// TIA Portal V15.1 export
// export: Created 2024-05-17T05:38:34.4008009Z, ExportSetting WithDefaults, DisplayName Totally Integrated Automation Portal, DisplayVersion V15.1 Update 5, DisplayName TIA Portal Openness, DisplayVersion V15.1 Update 5, DisplayName SINAMICS Startdrive Advanced, DisplayVersion V15.1, DisplayName G130, G150, S120, S150, SINAMICS MV, S210, DisplayVersion V15.1, DisplayName G110M, G120, G120C, G120D, G120P, DisplayVersion V15.1, DisplayName STEP 7 Professional, DisplayVersion V15.1 Update 5, DisplayName STEP 7 Safety, DisplayVersion V15.1, DisplayName WinCC Professional, DisplayVersion V15.1 Update 5, DisplayName SIMATIC Visualization Architect, DisplayVersion V15.1
FUNCTION_BLOCK "LProcSel5SP"   // FB1712, FBD
TITLE = LProcSel5SP
{ S7_Optimized_Access := 'FALSE' }
AUTHOR : VCC
FAMILY : ProcEq
NAME : Sel5SP
VERSION : 0.1
// ================================================================================
// This makes the selection of one set-point among 5 in function of the production 
// modes.
// The selection is made via a set-point request integer from 1 to 5.
// An external value is possible to be selected to set-point 1.
// ================================================================================
// stored: AutoNumber false, IsIECCheckEnabled false, SetENOAutomatically False, UDAEnableTagReadback false
   VAR_INPUT
      I_ExtSP1_Value { ExternalAccessible := 'False'; ExternalVisible := 'False'; ExternalWritable := 'False'} : Real;   // External Set-point 1
      H_SP2 : Real;   // Set-point 2
      H_SP3 : Real;   // Set-point 3
      H_SP4 : Real;   // Set-point 4
      H_SP5 : Real;   // Set-point 5
      I_SPReq : Int;   // Index Set-point Request
      I_ExtSP1 : Bool;   // External Set-point 1 Request
   END_VAR
   VAR_OUTPUT
      O_SPSel : Real;   // Set-point selected
   END_VAR
   VAR_IN_OUT
      H_SP1 : Real;   // Set-point 1
   END_VAR
BEGIN

REGION Network 1: **** 5.2 - Equations - Flow Equations **** Selection Set-point 1
   // Selection Set-point 1
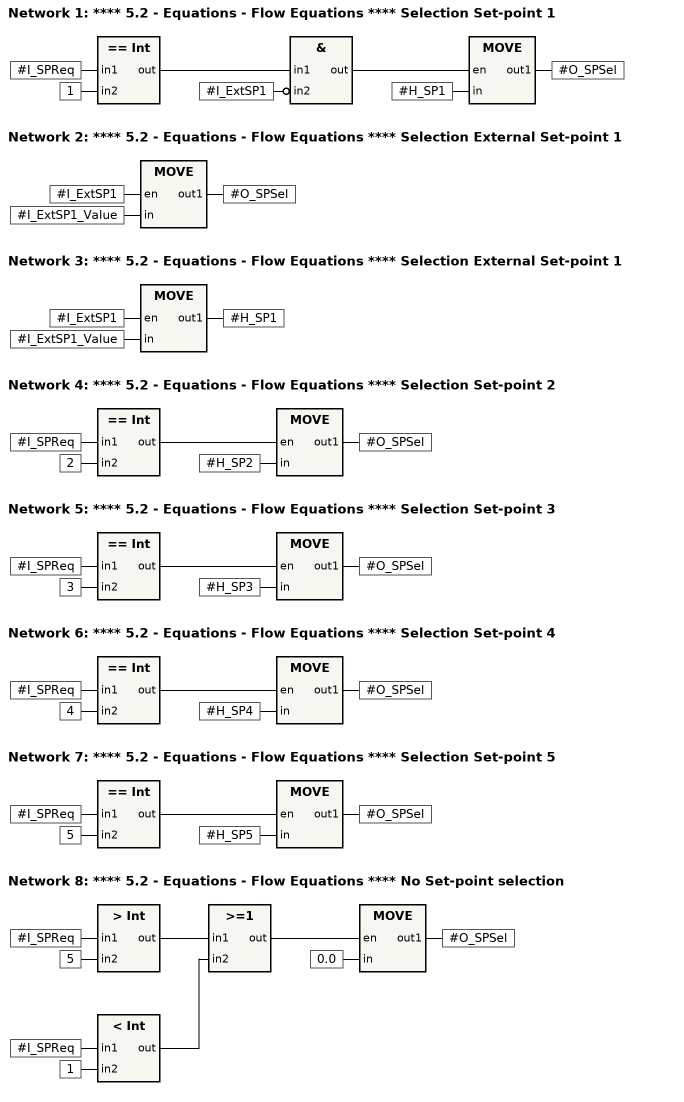
   IF (#I_SPReq = 1) AND NOT #I_ExtSP1 THEN #O_SPSel := #H_SP1; END_IF;
END_REGION

REGION Network 2: **** 5.2 - Equations - Flow Equations **** Selection External Set-point 1
   // Selection External Set-point 1
   IF #I_ExtSP1 THEN #O_SPSel := #I_ExtSP1_Value; END_IF;
END_REGION

REGION Network 3: **** 5.2 - Equations - Flow Equations **** Selection External Set-point 1
   // Selection External Set-point 1
   IF #I_ExtSP1 THEN #H_SP1 := #I_ExtSP1_Value; END_IF;
END_REGION

REGION Network 4: **** 5.2 - Equations - Flow Equations **** Selection Set-point 2
   // Selection Set-point 2
   IF #I_SPReq = 2 THEN #O_SPSel := #H_SP2; END_IF;
END_REGION

REGION Network 5: **** 5.2 - Equations - Flow Equations **** Selection Set-point 3
   // Selection Set-point 3
   IF #I_SPReq = 3 THEN #O_SPSel := #H_SP3; END_IF;
END_REGION

REGION Network 6: **** 5.2 - Equations - Flow Equations **** Selection Set-point 4
   // Selection Set-point 4
   IF #I_SPReq = 4 THEN #O_SPSel := #H_SP4; END_IF;
END_REGION

REGION Network 7: **** 5.2 - Equations - Flow Equations **** Selection Set-point 5
   // Selection Set-point 5
   IF #I_SPReq = 5 THEN #O_SPSel := #H_SP5; END_IF;
END_REGION

REGION Network 8: **** 5.2 - Equations - Flow Equations **** No Set-point selection
   // No Set-point selection
   IF (#I_SPReq > 5) OR (#I_SPReq < 1) THEN #O_SPSel := 0.0; END_IF;
END_REGION
END_FUNCTION_BLOCK
